// TIA Portal V17 export
// export: Created 2025-01-15T11:40:04.802159Z, ExportSetting WithDefaults, DisplayName Totally Integrated Automation Portal, DisplayVersion V17 Update 6, DisplayName TIA Portal Openness, DisplayVersion V17 Update 6, DisplayName TIA Portal Version Control Interface, DisplayVersion V17, DisplayName SINAMICS Startdrive Advanced, DisplayVersion V17 SP1, DisplayName SINAMICS Startdrive G130, G150, S120, S150, SINAMICS MV, S210, DisplayVersion V17 SP1, DisplayName SINAMICS Startdrive G110M, G120, G120C, G120D, G120P, G115D, DisplayVersion V17 SP1, DisplayName STEP 7 Professional, DisplayVersion V17 Update 6, DisplayName SINUMERIK ONE STEP 7 Toolbox, DisplayVersion V17 Update 2, DisplayName SINUMERIK 840D sl STEP 7 Toolbox, DisplayVersion V17 Update 2, DisplayName STEP 7 Safety, DisplayVersion V17 Update 6, DisplayName WinCC Advanced / Unified PC, DisplayVersion V17 Update 6
DATA_BLOCK "FB_SCL_Operations_DB"   // DB3
VERSION : 0.1
// stored: AutoNumber true, DBAccessibleFromOPCUA true, DBAccessibleFromWebserver true, InstanceOfName FB_SCL_Operations, InstanceOfType FB
"FB_SCL_Operations"
   // VAR_INPUT
   //    iBool : Bool;
   //    iInt_1 : Int;
   //    iInt_2 : Int;
   // END_VAR
   // VAR_OUTPUT
   //    qBool : Bool;
   //    qInt : Int;
   //    qIntDiv : Int;
   // END_VAR
BEGIN
END_DATA_BLOCK
